TYPE ST_DefaultEventClasses :
STRUCT
	Info,
	Warning,
	Error : TcEventEntry;
END_STRUCT
END_TYPE

(* stored: Version 1.1.0.1
   DUT ST_DefaultEventClasses: Id {accd1050-8a50-4afd-818c-0c8ad6b06666} *)
